// TwinCAT 3 PLC project Jenkins_CICD
// ProgramVersion: 3.1.4023.0
// project tree:
//   / FirstApp.TcPOU

// ---- FirstApp.TcPOU
PROGRAM FirstApp
VAR
	bIN: BOOL;
	bOut: BOOL;
END_VAR

bOut := bIN;

END_PROGRAM
